// Mitsubishi GX Developer project: Mitsubishi_Traffic_Light_4-road_junction   PLC: FX1S

PROGRAM MAIN
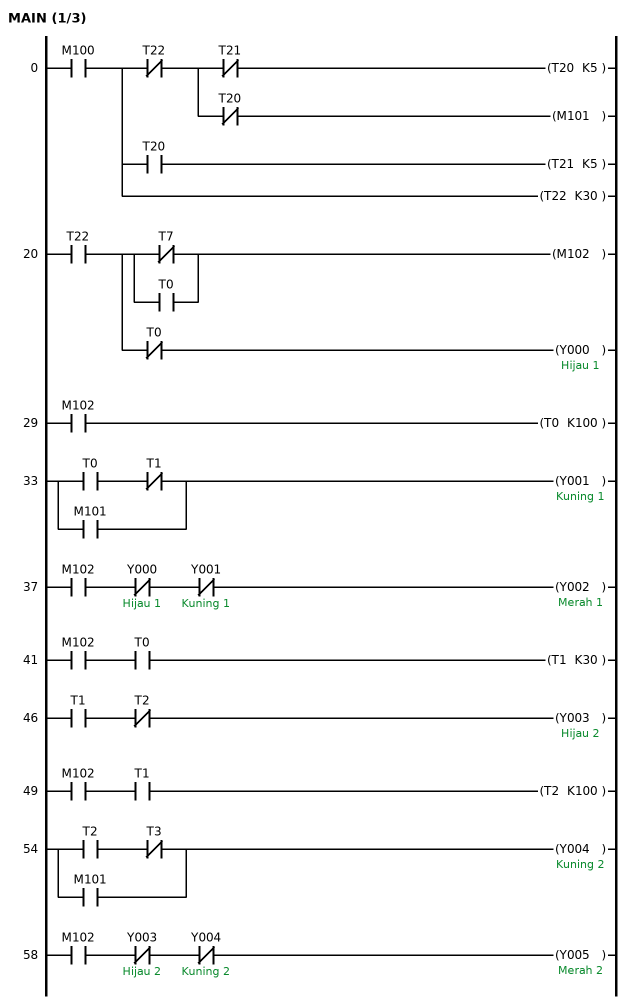
0     LD      M100
      MPS
      ANI     T22
      MPS
      ANI     T21
      OUT     T20 K5
      MPP
      ANI     T20
      OUT     M101
      MRD
      AND     T20
      OUT     T21 K5
      MPP
      OUT     T22 K30
20    LD      T22
      MPS
      LDI     T7
      OR      T0
      ANB
      OUT     M102
      MPP
      ANI     T0
      OUT     Y000  ; Hijau 1
29    LD      M102
      OUT     T0 K100
33    LD      T0
      ANI     T1
      OR      M101
      OUT     Y001  ; Kuning 1
37    LD      M102
      ANI     Y000  ; Hijau 1
      ANI     Y001  ; Kuning 1
      OUT     Y002  ; Merah 1
41    LD      M102
      AND     T0
      OUT     T1 K30
46    LD      T1
      ANI     T2
      OUT     Y003  ; Hijau 2
49    LD      M102
      AND     T1
      OUT     T2 K100
54    LD      T2
      ANI     T3
      OR      M101
      OUT     Y004  ; Kuning 2
58    LD      M102
      ANI     Y003  ; Hijau 2
      ANI     Y004  ; Kuning 2
      OUT     Y005  ; Merah 2
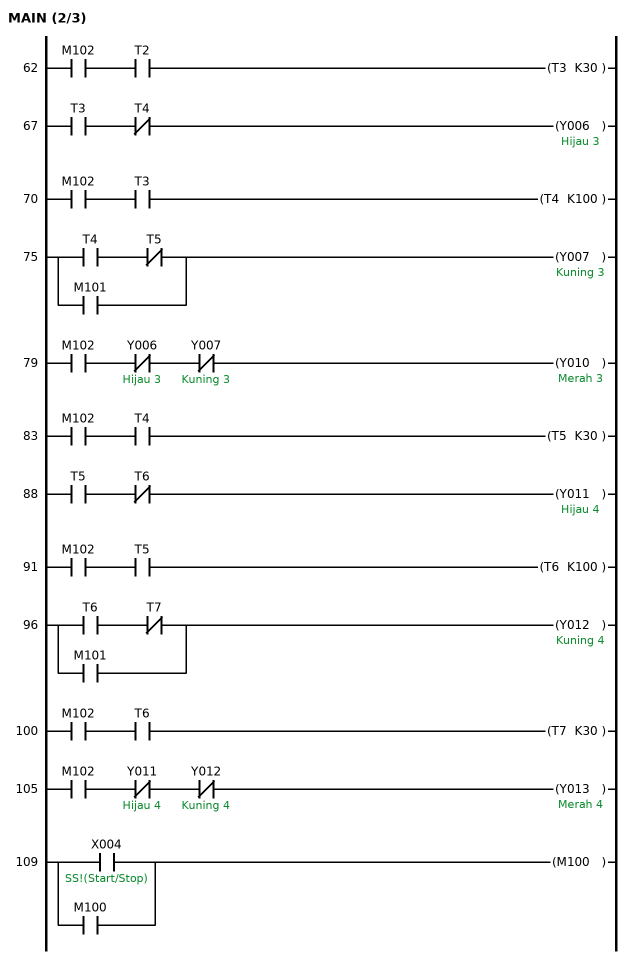
62    LD      M102
      AND     T2
      OUT     T3 K30
67    LD      T3
      ANI     T4
      OUT     Y006  ; Hijau 3
70    LD      M102
      AND     T3
      OUT     T4 K100
75    LD      T4
      ANI     T5
      OR      M101
      OUT     Y007  ; Kuning 3
79    LD      M102
      ANI     Y006  ; Hijau 3
      ANI     Y007  ; Kuning 3
      OUT     Y010  ; Merah 3
83    LD      M102
      AND     T4
      OUT     T5 K30
88    LD      T5
      ANI     T6
      OUT     Y011  ; Hijau 4
91    LD      M102
      AND     T5
      OUT     T6 K100
96    LD      T6
      ANI     T7
      OR      M101
      OUT     Y012  ; Kuning 4
100   LD      M102
      AND     T6
      OUT     T7 K30
105   LD      M102
      ANI     Y011  ; Hijau 4
      ANI     Y012  ; Kuning 4
      OUT     Y013  ; Merah 4
109   LD      X004  ; SS!(Start/Stop)
      OR      M100
      OUT     M100
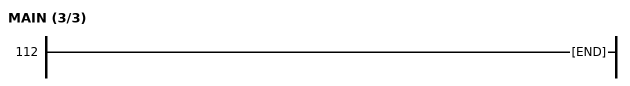
112   END
END_PROGRAM
